# B&R Automation Studio project SiemensBRCommunication
Automation Studio 4.10.2.37; technology packages: mapp 5.12.1, mappView 5.12.1

## Configuration Config2

CPU X20CP1584, AutomationRuntime B4.91, Build 4.1.2, Safety 0.0, Vc V4.72.2

### Task classes (Cpu.sw)
```
Cyclic#4:
  Com <- Com.prg
DataObjects: comDAVCfg <- comDAVCfg.dob, comDAVMap <- comDAVMap.dob
Binaries: FWRules, udbdef, TCData, mvLoader, arconfig, User, Role, iomap, asfw, ashwac, ashwd, sysconf, vcgclass, arsvcreg
Libraries: AsTCP, sys_lib, dvframe, asstring, runtime, standard, AsMem, AsIecCon, astime, DAVNoDave, arssl, fileio, dataobj, vcresman, aruser
```

### Hardware
```
X20CP1584 : X20CP1584 v1.9.0.0
  Connector IF2:
    ActivateDevice = 1
    Mode = Manual
    InternetAddress = 192.168.0.3
    SubnetMask = 255.255.255.0
  Connector IF3:
    Operation = EthOnly
    EthernetMode = Manual
    InternetAddress = 10.42.10.220
    SubnetMask = 255.255.255.0
  ConfigurationID = komunikaceSIMATIC_Config2
  UserPartitionSize = 100
  AutomaticTransferOfUserfiles = on
  FileDevice1
  FileDeviceName1 = Flashcard
  FileDevicePath1 = C:\
  FtpUser1
  FtpUsername1 = admin
  FtpUserPassword1 = b1OGEwZ56wPH8RQzCv5cMjA1xEZ3AQeIlDvIGC2uv18=
  FtpUserSalt1 = TsE2z1/6
  FTPAccessRight1 = 0
  FTPdevice1 = ALL
  ActivateOpcUa = 1
  OpcUaInformationModels_PV_Version = 1
```

## Logical view

Binary libraries used (declarations not repeated): AsTCP, sys_lib, dvframe, asstring, runtime, standard, AsMem, AsIecCon, astime, DataObj

### Global.typ - Global data types
```iecst
TYPE
	comunicationStatus :
		(
		Initializing,
		Connecting,
		Connected,
		Disconnecting,
		Disconected,
		InitializationError,
		ConnectionError,
		ClientError,
		DisconnectingError
	);
END_TYPE
```

### Package Logical/Libraries - Global libraries

### Library Logical/Libraries/DAVNoDave (IEC, version 1.04.0) - A library based on LibNoDave to connect to a Siemens PLC
Depends on: AsTCP, DataObj, sys_lib, dvframe, asstring

#### DAVNoDave.fun - Exported functions and function blocks
```iecst
(********************************************************************
 * COPYRIGHT -- B&R Industrial Automation
 ********************************************************************
 * Library: DAVNoDave
 * File: DAVNoDave.fun
 * Author: morrisd
 * Created: May 26, 2009
 ********************************************************************
 * Functions and function blocks of library DAVNoDave
 ********************************************************************)
(**)
(*Initialization*)

FUNCTION_BLOCK DAVinitialize (*Allocates memory for communications*)
	VAR_INPUT
		enable : BOOL; (*Enable function block*)
		reset : BOOL; (*Resets the function block in case of error or if you want to reload the dataobjects ...*)
		pDOConfig : UDINT; (*Address of the name of the data object used for configuration*)
		pDOMapping : UDINT; (*Address of the name of the data object used for variable mapping*)
		pMemIdent : UDINT; (*Pointer to memory allocated by user in InitUp*)
		numItemsConfig : UINT; (*Maximum number of items in the configuration data object*)
		numItemsMapping : UINT; (*Maximum number of items in the mapping data object*)
	END_VAR
	VAR_OUTPUT
		status : UINT; (*Function block status*)
		handle : UDINT; (*Handle (for other functions)*)
	END_VAR
	VAR
		state : USINT;
		pConfig : REFERENCE TO DAVConfig_typ;
		pConfigSwap : REFERENCE TO DAVConfig_typ;
		pMapping : REFERENCE TO DAVMapping_typ;
		pMappingSwap : REFERENCE TO DAVMapping_typ;
		pDAV : REFERENCE TO DAVHandle_typ;
		pData : REFERENCE TO ARRAY[0..499] OF USINT;
		DatObjInfo_Config : DatObjInfo;
		DatObjInfo_Map : DatObjInfo;
		DatObjRead_0 : DatObjRead;
		charIdx : UDINT;
		configIdx : UINT;
		configTemp : DAVConfig_typ;
		orderIdx : UINT;
		scanCount : UDINT;
		curDataLength : UDINT;
		status_i : UINT;
		curVarType : UDINT;
		curDimensions : UDINT;
		mappingTemp : DAVMapping_typ;
		lengthToAllocate : UDINT;
		pDOData : UDINT;
		mappingIdx : UINT;
		straSplit : ARRAY[0..9] OF STRING[100];
		posNextNull : UINT;
		tmpAdr : UDINT;
		tmpVal : DINT;
		posPlus : UINT;
		memFreeFB : {REDUND_UNREPLICABLE} ARRAY[0..1] OF AsMemPartFree;
		memAllocFB : {REDUND_UNREPLICABLE} ARRAY[0..1] OF AsMemPartAllocClear;
		memHandle : {REDUND_UNREPLICABLE} ARRAY[0..1] OF UDINT;
		i : {REDUND_UNREPLICABLE} USINT;
	END_VAR
END_FUNCTION_BLOCK
(**)
(*Connection*)

FUNCTION_BLOCK DAVconnect (*Connects to a Siemens S7 or VIPA unit via ISO/TCP*)
	VAR_INPUT
		enable : BOOL; (*Enable function block*)
		pHandle : UDINT; (*Address of handle from DAVinitialize*)
		protocol : USINT; (*Connection mode. Use DAV_PROTOCOL_xxx*)
		pMPIinterface : UDINT; (*MPI interface to use (i.e. 'IF1')*)
		pMPIconnection : UDINT; (*MPI connection parameters. Use 0 for DAV_DEFAULT_MPI*)
		MPIspeed : USINT; (*MPI speed. Use DAV_SPEED_xxx*)
		MPIlocalAdr : USINT; (*MPI local address. Usually 1*)
		MPIplcAdr : USINT; (*MPI PLCl address. Usually 2*)
		pTCPsourceIP : UDINT; (*TCP ethernet interface - use 0 for listenning in on all interfaces.*)
		pTCPtargetIP : UDINT; (*TCP IP address to connect to*)
		TCPport : UINT; (*TCP port to use - use 0 for DAV_DEFAULT_PORT*)
		TCPrack : USINT; (*TCP rack number (usually 0)*)
		TCPslot : USINT; (*TCP slot number (usually 1)*)
		timeout : UINT; (*Timout time*)
	END_VAR
	VAR_OUTPUT
		status : UINT; (*Function block status*)
		pduLength : UINT; (*Length of PDU (from PLC)*)
		portOpened : UINT; (*Port number used for connection*)
		TCPident : UDINT;
	END_VAR
	VAR
		pDAV : REFERENCE TO DAVHandle_typ;
		pBufferR : REFERENCE TO ARRAY[0..99] OF USINT;
		state : USINT;
		frmConfig : XOPENCONFIG;
		FRM_xopen_0 : FRM_xopen;
		TcpOpen_0 : TcpOpen;
		TcpClient_0 : TcpClient;
		DAVexchange_0 : DAVexchange;
		TON_10ms_ClientTimeout : TON_10ms;
	END_VAR
END_FUNCTION_BLOCK

FUNCTION_BLOCK DAVdisconnect (*Disconnects current connection*)
	VAR_INPUT
		enable : BOOL; (*Enable function block*)
		pHandle : UDINT; (*Address of handle from DAVinitialize*)
		timeout : UINT;
	END_VAR
	VAR_OUTPUT
		status : UINT; (*Function block status*)
	END_VAR
	VAR
		pDAV : REFERENCE TO DAVHandle_typ;
		TcpClose_0 : TcpClose;
		FRM_close_0 : FRM_close;
		DAVexchange_0 : DAVexchange;
		state : USINT;
	END_VAR
END_FUNCTION_BLOCK
(**)
(*Servicing*)

FUNCTION_BLOCK DAVclient (*Services communcations between a B&R and Siemens PLC*)
	VAR_INPUT
		enable : BOOL; (*Enable function block*)
		pHandle : UDINT; (*Address of handle from DAVinitialize*)
		pause : BOOL; (*Pause the data transfer*)
		timeout : UINT; (*Timeout when reading*)
	END_VAR
	VAR_OUTPUT
		status : UINT; (*Function block status*)
		paused : BOOL; (*Whether the communications have been paused*)
		errorPackets : UINT; (*Number of misconfigured packets*)
		safeToDisconnect : BOOL; (*TRUE when the user can disconnect*)
	END_VAR
	VAR
		state : USINT;
		pDAV : REFERENCE TO DAVHandle_typ;
		pConfig : REFERENCE TO DAVConfig_typ;
		pMapping : REFERENCE TO DAVMapping_typ;
		ppBuffer : REFERENCE TO ARRAY[0..499] OF USINT;
		DAVexchange_0 : DAVexchange;
		currentMode : USINT;
		currentPriority : USINT;
		addIdx : UINT;
		findIdx : USINT;
		itemIdx : UINT;
		mapIdx : UINT;
		readIdx : UINT;
		numItems : USINT;
		varList : ARRAY[0..19] OF UINT;
		curValue : UDINT;
		dataLength : UINT;
		bufferFull : BOOL;
		moreLinesToScan : BOOL;
		writeValues : ARRAY[0..19] OF UDINT;
		responseSize : UINT;
		numItemsCfg : USINT;
		numItemsMap : USINT;
		maxSendSize : UINT;
		useVariable : BOOL;
		pEnable : REFERENCE TO BOOL;
	END_VAR
END_FUNCTION_BLOCK
(**)
(*Internal - Data exchange*)

FUNCTION_BLOCK DAVexchange (*Exchanges data between PLC's*)
	VAR_INPUT
		enable : BOOL; (*Enable function block*)
		pHandle : UDINT; (*Address of handle from DAVinitialize*)
		sendLength : UINT; (*Length of data to send*)
		timeout : UINT; (*Timeout when reading*)
		mpiFullExchange : BOOL; (*Full exchange of data, including Acknowledges. MPI protocol only*)
	END_VAR
	VAR_OUTPUT
		status : UINT; (*Function block status*)
		recvLength : UINT; (*Received number of bytes (not including header)*)
		recvParamLength : UINT; (*Length of parameter area*)
		recvDataLength : UINT; (*Length of data area*)
		recvStartOfDataIdx : UINT; (*Number of bytes (index 0) before data starts*)
	END_VAR
	VAR
		state : USINT;
		pDAV : REFERENCE TO DAVHandle_typ;
		ppBuffer : REFERENCE TO ARRAY[0..19] OF USINT;
		TcpSend_0 : TcpSend;
		TcpRecv_0 : TcpRecv;
		TON_10ms_Timeout : TON_10ms;
		DAVmpiSend_0 : DAVmpiSend;
		DAVmpiRead_0 : DAVmpiRead;
		bufferRead : ARRAY[0..19] OF USINT;
		bufferSend : ARRAY[0..19] OF USINT;
		sendAckNumber : USINT;
		lastState : USINT;
	END_VAR
END_FUNCTION_BLOCK

FUNCTION_BLOCK DAVmpiSend (*Sends data via serial (DVFrame library)*)
	VAR_INPUT
		enable : BOOL; (*Enable function block*)
		ident : UDINT; (*Ident from FRM_Xopen*)
		sendLength : UINT; (*Length to send*)
		pBufferW : UDINT; (*Pointer to data to send*)
	END_VAR
	VAR_OUTPUT
		status : UINT; (*Function block status*)
	END_VAR
	VAR
		FRM_gbuf_0 : FRM_gbuf;
		FRM_write_0 : FRM_write;
		FRM_robuf_0 : FRM_robuf;
	END_VAR
END_FUNCTION_BLOCK

FUNCTION_BLOCK DAVmpiRead (*Reads data via serial (DVFrame library)*)
	VAR_INPUT
		enable : BOOL; (*Enable function block*)
		ident : UDINT; (*Ident from FRM_Xopen*)
		pBufferR : UDINT; (*Maximum length to read*)
		readLength : UINT; (*Pointer to storage to read data into*)
	END_VAR
	VAR_OUTPUT
		status : UINT; (*Function block status*)
		recvBufferLength : UINT;
	END_VAR
	VAR
		FRM_read_0 : FRM_read;
		FRM_rbuf_0 : FRM_rbuf;
	END_VAR
END_FUNCTION_BLOCK
(**)
(*Internal - Packets*)

FUNCTION DAVpacketHeader : UINT (*Initializes a packet with the required protocol and TPDU. Returns the index to the start of the TPDU*)
	VAR_INPUT
		pDAV : REFERENCE TO DAVHandle_typ; (*Pointer to DAVHandle_typ*)
		pBuffer : REFERENCE TO ARRAY[0..19] OF USINT; (*Pointer to buffer to build the message*)
	END_VAR
END_FUNCTION

FUNCTION DAVpacketReadInit : UINT (*Initializes a packet for writing variables. Returns number of bytes in the buffer*)
	VAR_INPUT
		pDAV : REFERENCE TO DAVHandle_typ; (*Pointer to DAVHandle_typ*)
		pBuffer : REFERENCE TO ARRAY[0..19] OF USINT; (*Pointer to buffer to build the message*)
	END_VAR
END_FUNCTION

FUNCTION DAVpacketReadAddVar : UINT (*Adds a variable to a read packet. Returns number of bytes in the buffer*)
	VAR_INPUT
		pDAV : REFERENCE TO DAVHandle_typ; (*Pointer to DAVHandle_typ*)
		pBuffer : REFERENCE TO ARRAY[0..19] OF USINT; (*Pointer to buffer to build the message*)
		pVar : REFERENCE TO DAVSendVar_typ; (*Pointer to variable configuration to use*)
	END_VAR
	VAR
		ppBuffer : REFERENCE TO ARRAY[0..12] OF USINT;
		packetLength : UINT;
		paramLength : UINT;
	END_VAR
END_FUNCTION

FUNCTION DAVpacketWriteInit : UINT (*Initialiizes a packet for writing variables. Returns number of bytes in the buffer*)
	VAR_INPUT
		pDAV : REFERENCE TO DAVHandle_typ; (*Pointer to DAVHandle_typ*)
		pBuffer : REFERENCE TO ARRAY[0..19] OF USINT; (*Pointer to buffer to build the message*)
	END_VAR
END_FUNCTION

FUNCTION DAVpacketWriteAddVar : UINT (*Adds a variable to a write packet. Returns number of bytes in the buffer*)
	VAR_INPUT
		pDAV : REFERENCE TO DAVHandle_typ; (*Pointer to DAVHandle_typ*)
		pBuffer : REFERENCE TO ARRAY[0..19] OF USINT; (*Pointer to buffer to build the message*)
		pWriteBuffer : REFERENCE TO ARRAY[0..3] OF USINT; (*Pointer to write data*)
		pVar : REFERENCE TO DAVSendVar_typ; (*Pointer to variable configuration to use*)
	END_VAR
	VAR
		ppBuffer : REFERENCE TO ARRAY[0..12] OF USINT;
		packetLength : UINT;
		paramLength : UINT;
		dataLength : UINT;
		pBufferData : UDINT;
	END_VAR
END_FUNCTION

FUNCTION DAVpacketTCPconnect : UINT (*Creates packets for establishing a connection to a PLC via ISO/TCP. Returns number of bytes in the buffer*)
	VAR_INPUT
		pDAV : REFERENCE TO DAVHandle_typ; (*Pointer to DAVHandle_typ*)
		pBuffer : REFERENCE TO ARRAY[0..25] OF USINT; (*Pointer to buffer to build the message*)
		num : USINT; (*Packet to create*)
	END_VAR
END_FUNCTION

FUNCTION DAVpacketMPIconnect : UINT (*Creates packets for establishing a connection to a PLC via MPI. Returns number of bytes in the buffer*)
	VAR_INPUT
		pDAV : REFERENCE TO DAVHandle_typ; (*Pointer to DAVHandle_typ*)
		pBuffer : REFERENCE TO ARRAY[0..49] OF USINT; (*Pointer to buffer to build the message*)
		num : USINT; (*Packet to create*)
	END_VAR
END_FUNCTION

FUNCTION DAVpacketMPIdisconnect : UINT (*Creates packets for disconnect from a PLC via MPI. Returns number of bytes in the buffer*)
	VAR_INPUT
		pDAV : REFERENCE TO DAVHandle_typ; (*Pointer to DAVHandle_typ*)
		pBuffer : REFERENCE TO ARRAY[0..19] OF USINT; (*Pointer to buffer to build the message*)
		num : USINT; (*Packet to create*)
	END_VAR
END_FUNCTION

FUNCTION DAVpacketMPIack : UINT (*Creates packets for sending an Acknowledge to a PLC via MPI. Returns number of bytes in the buffer*)
	VAR_INPUT
		pDAV : REFERENCE TO DAVHandle_typ; (*Pointer to DAVHandle_typ*)
		pBuffer : REFERENCE TO ARRAY[0..11] OF USINT; (*Pointer to buffer to build the message*)
		ackNum : USINT; (*Acknowledge number to use*)
	END_VAR
END_FUNCTION

FUNCTION DAVresponseMPIconnect : UINT (*Compares the response of a packet from the PLC with what is expected. Returns if the packet is okay*)
	VAR_INPUT
		pDAV : REFERENCE TO DAVHandle_typ; (*Pointer to DAVHandle_typ*)
		pBuffer : REFERENCE TO ARRAY[0..49] OF USINT; (*Pointer to buffer to compare the message*)
		num : USINT; (*Packet to compare*)
	END_VAR
END_FUNCTION
(**)
(*Internal - Swap bytes*)

FUNCTION DAVswapWORD : UINT (*Swaps bytes in a WORD*)
	VAR_INPUT
		pUINT : REFERENCE TO UINT; (*Address of UINT variable*)
	END_VAR
END_FUNCTION

FUNCTION DAVswapDWORD : UDINT (*Swaps bytes and words in a DWORD*)
	VAR_INPUT
		pUDINT : REFERENCE TO UDINT; (*Address of UDINT variable*)
	END_VAR
END_FUNCTION
(**)
(*Internal - Get bytes*)

FUNCTION DAVgetHIBYTE : USINT (*Returns the hi-byte from a WORD*)
	VAR_INPUT
		input : UINT; (*Input WORD*)
	END_VAR
END_FUNCTION

FUNCTION DAVgetLOBYTE : USINT (*Returns the lo-byte from a WORD*)
	VAR_INPUT
		input : UINT; (*Input WORD*)
	END_VAR
END_FUNCTION

FUNCTION DAVaddressBITS : USINT (*Returns a byte of the start address*)
	VAR_INPUT
		startAdr : UDINT; (*Start address of variable*)
		byteNum : USINT; (*Byte number to return*)
	END_VAR
END_FUNCTION
(**)
(*Internal - Combine bytes*)

FUNCTION DAVmakeWORD : UINT (*Returns a WORD from 2 bytes*)
	VAR_INPUT
		hiByte : USINT; (*Hi-byte input*)
		loByte : USINT; (*Lo-byte input*)
	END_VAR
END_FUNCTION

FUNCTION DAVupdateVAR : USINT (*Updates the selected variable*)
	VAR_INPUT
		pMapping : REFERENCE TO DAVMapping_typ; (*Pointer to a DAVMapping_typ*)
		pBuffer : UDINT; (*Address of buffer to read the value*)
		transportBOOL : BOOL; (*Transport mechanism for BOOLEAN data*)
	END_VAR
	VAR
		pDynBool : REFERENCE TO BOOL;
		pDynByte : REFERENCE TO USINT;
		pDynWord : REFERENCE TO UINT;
		pDynDWord : REFERENCE TO UDINT;
		tempVar : UDINT;
	END_VAR
END_FUNCTION

FUNCTION DAVcalcVARadr : USINT
	VAR_INPUT
		pVar : REFERENCE TO DAVSendVar_typ; (*Pointer to DAVSendVar_typ*)
	END_VAR
	VAR
		pUserDB : REFERENCE TO UINT;
		pUserStartAdr : REFERENCE TO UINT;
		pUserStartAdrB : REFERENCE TO USINT;
	END_VAR
END_FUNCTION
(**)
(*Internal - Misc*)

FUNCTION DAVsplit : UINT
	VAR_INPUT
		pData : UDINT; (*Address of data to read*)
		pSplitData : REFERENCE TO ARRAY[0..9] OF STRING[100]; (*Pointer to array of strings*)
	END_VAR
	VAR
		ppData : REFERENCE TO ARRAY[0..499] OF USINT;
		ppSplitData : REFERENCE TO ARRAY[0..99] OF USINT;
		splitIdx : USINT;
		charIdx : UINT;
		copyIdx : UINT;
	END_VAR
END_FUNCTION

FUNCTION DAVisnumeric : BOOL
	VAR_INPUT
		pString : UDINT; (*Pointer to string to compare*)
	END_VAR
	VAR
		pData : REFERENCE TO ARRAY[0..99] OF USINT;
		charIdx : USINT;
	END_VAR
END_FUNCTION

FUNCTION DAVmpiCalcCS : BOOL
	VAR_INPUT
		pBuffer : REFERENCE TO ARRAY[0..99] OF USINT; (*Address of buffer*)
		len : UINT; (*Length to data*)
	END_VAR
	VAR
		charIdx : UINT;
		checksum : USINT;
	END_VAR
END_FUNCTION

FUNCTION DAVmpiSuffixCRC : UINT (*Performs DLE doubling, adds DLE and ETX and BCC (checksum)*)
	VAR_INPUT
		pBuffer : REFERENCE TO ARRAY[0..499] OF USINT; (*Pointer to buffer to build the message*)
		len : UINT; (*Length of data in the buffer*)
	END_VAR
	VAR
		bufferR : ARRAY[0..499] OF USINT;
		sourceIdx : UINT;
		destIdx : UINT;
		bcc : USINT;
	END_VAR
END_FUNCTION

FUNCTION DAVdecodeMPI : UINT (*Removes DLE doubling from a received message*)
	VAR_INPUT
		pBuffer : REFERENCE TO ARRAY[0..499] OF USINT; (*Pointer to buffer which contains the message*)
		bufferSize : UINT; (*Total size of the buffer*)
		dataLength : UINT; (*Length of data currently in the buffer*)
	END_VAR
	VAR
		bufferOrig : ARRAY[0..499] OF USINT;
		sourceIdx : UINT;
		destIdx : UINT;
	END_VAR
END_FUNCTION
```

#### DAVNoDave.typ - Exported data types
```iecst
(********************************************************************
 * COPYRIGHT -- B&R Industrial Automation
 ********************************************************************
 * Library: DAVNoDave
 * File: DAVNoDave.typ
 * Author: morrisd
 * Created: May 26, 2009
 ********************************************************************
 * Functions and function blocks of library DAVNoDave
 ********************************************************************)
(**)
(*DAV Handle*)

TYPE
	DAVHandle_typ : 	STRUCT  (*Main DAVNoDave structure*)
		connection : DAVHandleConnect_typ; (*Connection data*)
		ident : UDINT; (*Identity for TCP / MPI comms*)
		pConfig : UDINT; (*Address of comms configuration*)
		pMapping : UDINT; (*Address of mapping configuration*)
		pBufferR : UDINT; (*Address of read buffer*)
		pBufferW : UDINT; (*Address of write buffer*)
		internal : USINT; (*Internal*)
		maxLinesConfig : UINT; (*Maximum number of lines in configuration*)
		maxLinesMapping : UINT; (*Maximum number of lines in mapping*)
		maxPrioirty : USINT; (*Maximum prioirty level found in the configuration data object*)
	END_STRUCT;
	DAVHandleConnect_typ : 	STRUCT  (*DAVNoDave communications*)
		protocol : USINT; (*Protocol (DAV_PROTOCOL_xxx)*)
		mpiSpeed : USINT; (*MPI speed (DAV_SPEED_xxx)*)
		mpiLocalAdr : USINT; (*MPI local address (usually 1)*)
		mpiPLCAdr : USINT; (*MPI PLC address (usually 2)*)
		tcpRack : USINT; (*TCP rack*)
		tcpSlot : USINT; (*TCP slot*)
		connectNum : USINT; (*MPI connection number*)
		connectNum2 : USINT; (*MPI connection number 2*)
		msgNum : USINT; (*Packet number*)
		pduNum : UINT; (*PDU number*)
		ackNum : USINT; (*Acknowledge number*)
	END_STRUCT;
END_TYPE

(**)
(*Data Object (per line)*)

TYPE
	DAVSendVar_typ : 	STRUCT  (*Structure per variable per variable*)
		area : USINT; (*Siemens - Area (DAV_AREA_xxx)*)
		db : UINT; (*Siemens - Data block number (only if area is DAV_AREA_DB)*)
		pdb : UDINT; (*Siemens - Pointer to Data block number (only if area is DAV_AREA_DB)*)
		actAdr : UINT; (*Siemens - Actual variable address (in BYTE's)*)
		bitAdr : UDINT; (*Siemens - Start address (in BIT's)*)
		pStartAdr : UDINT; (*Siemens - Pointer to Start address (must be a UINT)*)
		bitAdrB : USINT; (*Siemens - Start address bit position*)
		pStartAdrB : UDINT; (*Siemens - Pointer to start address bit position (must be a USINT)*)
		type : USINT; (*Siemens - Variable type (DAV_VAR_xxx)*)
		length : UINT; (*Siemens - Variable length*)
	END_STRUCT;
	DAVConfig_typ : 	STRUCT  (*Structure per line in the configuration data object*)
		var : DAVSendVar_typ; (*Variable details*)
		priority : USINT; (*Priority of variable*)
		pEnable : UDINT; (*Pointer to enable variable (must be a BOOL)*)
		brVarAdr : UDINT; (*B&R - Start address of variable(s)*)
		internal : USINT; (*Internal variable*)
	END_STRUCT;
	DAVMapping_typ : 	STRUCT  (*Structure per line in the mapping data object*)
		var : DAVSendVar_typ; (*Variable details*)
		priority : USINT; (*Priority of variable*)
		pEnable : UDINT; (*Pointer to enable variable (must be a BOOL)*)
		access : USINT; (*Access (0 = read, 1= write, 2 = both)*)
		brVarAdr : UDINT; (*B&R - Address of variable to store the value*)
		brVarLength : USINT; (*B&R - Length of variable*)
		brVarType : USINT; (*B&R - Variable type*)
		brPrevValue : UDINT; (*B&R - Previous value*)
		internal : USINT; (*Internal variable*)
		cfgIndex : UINT; (*Internal configuration index*)
	END_STRUCT;
END_TYPE
```

#### DAVNoDave.var - Exported constants
```iecst
(********************************************************************
 * COPYRIGHT -- B&R Industrial Automation
 ********************************************************************
 * Library: DAVNoDave
 * File: DAVNoDave.var
 * Author: morrisd
 * Created: May 26, 2009
 ********************************************************************
 * Constants of library DAVNoDave
 ********************************************************************)
(**)
(*Internal*)
VAR CONSTANT
	DAV_DEFAULT_BUFFER_R : UINT := 500; (*Default read buffer size, should be more than PDU size*)
	DAV_DEFAULT_BUFFER_W : UINT := 500; (*Default write buffer size, should be more than PDU size*)
END_VAR
(**)
(*Default values*)
VAR CONSTANT
	DAV_DEFAULT_SOURCE_PORT : UINT := 60000; (*Default source port (should be >=49152)*)
	DAV_DEFAULT_PORT : UINT := 102; (*Default connection port*)
	DAV_DEFAULT_MPI : STRING[40] := '/PHY=RS232 /BD=38400 /PA=O /DB=8 /SB=1'; (*Default connection for MPI*)
	DAV_DEFAULT_TIMEOUT : UINT := 0; (*Default timeout (1500ms for ISO/TCP, 5000ms for MPI)*)
END_VAR
(**)
(*Configuration*)
VAR CONSTANT
	DAV_CONFIG_MAX_LINES : UINT := 500; (*Maximum number of lines in the configuration file*)
	DAV_CONFIG_PRIOIRTY_MAX : USINT := 5; (*Prioirty level (maximum)*)
	DAV_CONFIG_RW_B : USINT := 2; (*Access level (read / write)*)
	DAV_CONFIG_RW_R : USINT := 1; (*Access level (read only)*)
	DAV_CONFIG_RW_W : USINT := 3; (*Access level (write only)*)
END_VAR
(**)
(*Protocol*)
VAR CONSTANT
	DAV_PROTOCOL_TCP : USINT := 100; (*Connection type - ISOTCP*)
	DAV_PROTOCOL_MPI : USINT := 200; (*Connection type - MPI*)
END_VAR
(**)
(*Protocol - Speed*)
VAR CONSTANT
	DAV_SPEED_9K : USINT := 0; (*MPI Adapter speed - 9k baud*)
	DAV_SPEED_19K : USINT := 1; (*MPI Adapter speed - 19k baud*)
	DAV_SPEED_187K : USINT := 2; (*MPI Adapter speed - 187k baud*)
	DAV_SPEED_500K : USINT := 3; (*MPI Adapter speed - 500k baud*)
	DAV_SPEED_1500K : USINT := 4; (*MPI Adapter speed - 1500k baud*)
	DAV_SPEED_45K : USINT := 5; (*MPI Adapter speed - 45k baud*)
	DAV_SPEED_93K : USINT := 6; (*MPI Adapter speed - 93k baud*)
END_VAR
(**)
(*PDU Constants*)
VAR CONSTANT
	DAV_PDU_SIZE : UINT := 240; (*PDU size*)
END_VAR
(**)
(*Variables*)
VAR CONSTANT
	DAV_VAR_BIT : USINT := 1; (*Read a single bit*)
	DAV_VAR_BYTE : USINT := 2; (*Read a byte*)
	DAV_VAR_WORD : USINT := 4; (*NOT IMPLEMENTED Read a word*)
END_VAR
(**)
(*DataBlock's and Area*)
VAR CONSTANT
	DAV_AREA_COUNTER : USINT := 28; (*NOT IMPLEMENTED Area type, S7 Counters*)
	DAV_AREA_DB : USINT := 132; (*Area type, DataBlocks*)
	DAV_AREA_DI : USINT := 133; (*NOT IMPLEMENTED Area type, DataBlock Instance*)
	DAV_AREA_FLAG : USINT := 131; (*Area type, Flags*)
	DAV_AREA_INPUT : USINT := 129; (*Area type, Inputs*)
	DAV_AREA_LOCAL : USINT := 134; (*NOT IMPLEMENTED Area type, Local (not tested)*)
	DAV_AREA_OUTPUT : USINT := 130; (*Area type, Outputs*)
	DAV_AREA_PERIPHERAL : USINT := 128; (*NOT IMPLEMENTED Area type, Peripherals*)
	DAV_AREA_TIMER : USINT := 29; (*NOT IMPLEMENTED Area type, S7 Timers*)
END_VAR
(**)
(*Error codes*)
VAR CONSTANT
	DAV_ERR_INITIALIZATION : UINT := 51000; (*Initialization error*)
	DAV_ERR_HANDLE : UINT := 51001; (*Invalid handle specified*)
	DAV_ERR_BUFFER : UINT := 51002; (*Invalid buffer specified*)
	DAV_ERR_BUFFER_SIZE : UINT := 51003; (*Invalid buffer size specified*)
	DAV_ERR_CONNECT_OPEN : UINT := 51004; (*Connection already open*)
	DAV_ERR_CONNECT_CLOSED : UINT := 51005; (*Connection already closed*)
	DAV_ERR_CONNECT_PROTOCOL : UINT := 51006; (*Invalid connection mode specidied*)
	DAV_ERR_CONNECT_TARGETIP : UINT := 51007; (*Invalid target IP specified*)
	DAV_ERR_CONNECT_INTERFACE : UINT := 51008; (*Invalid interface specified*)
	DAV_ERR_CONNECT_TCP : UINT := 51009; (*Can not connect to specified TCP/IP address*)
	DAV_ERR_SEND_MISSINGDATA : UINT := 51010; (*Not all the data was sent*)
	DAV_ERR_SEND_NODATA : UINT := 51011; (*Invalid send length*)
	DAV_ERR_SEND_BUFFERSIZE : UINT := 51012; (*Buffer size too small*)
	DAV_ERR_RECV_NODATA : UINT := 51020; (*No data received - client disconnect?*)
	DAV_ERR_RECV_MISSINGDATA : UINT := 51021; (*Not all the data was received*)
	DAV_ERR_RECV_WRONGPACKET : UINT := 51022; (*Wrong packet received*)
	DAV_ERR_RECV_BUFFERSIZE : UINT := 51023; (*Buffer size too small*)
	DAV_ERR_RECV_PROTOCOL : UINT := 51024; (*MPI protocol error*)
	DAV_ERR_RECV_RESPONSE : UINT := 51025; (*MPI response*)
	DAV_ERR_FAILED_READ : UINT := 51027; (*Failed to read data*)
	DAV_ERR_FAILED_WRITE : UINT := 51028; (*Failed to write data*)
	DAV_ERR_TIMEOUT : UINT := 51029; (*Timeout occured*)
	DAV_ERR_CFG_DONAME : UINT := 51030; (*Invalid configuration specified*)
	DAV_ERR_CFG_DONODATA : UINT := 51031; (*Invalid configuration data (none available)*)
	DAV_ERR_CFG_INVALID : UINT := 51032; (*Invalid configuration data*)
	DAV_ERR_CFG_MAXLINES : UINT := 51033; (*Invalid number of lines specified*)
	DAV_ERR_CFG_TIMEOUT : UINT := 51034; (*Execution too long*)
	DAV_ERR_MPI_ADAPTER : UINT := 51040; (*Unsupported MPI adapter*)
	DAV_ERR_ACKNOWLEDGE : UINT := 51041;
END_VAR
```

#### DAVinitialize.st - Initializes data object(s) for servicing communications
```iecst
(********************************************************************************************************************************)
(* COPYRIGHT -- B&R Industrial Automation																																												*)
(********************************************************************************************************************************)
(* Library:				DAVNoDave																																																			*)
(* File: 					DAVinitialize.st																																															*)
(* Author: 				morrisd																																																				*)
(* Created: 			May 26, 2009																																																	*)
(********************************************************************************************************************************)

(********************************************************************************************************************************)
(* DAVinitialize																																																								*)
(*==============================================================================================================================*)
(* Initializes the configuration object to communicate between the PLC and the Siemen's PLC																			*)
(* Note:																																																												*)
(*			1) This function needs to be called in the INIT program. 																																*)
(*			2) It should be called once and not continously in a loop (as we call it in a loop).																		*)
(* Returns a status																																																							*)
(********************************************************************************************************************************)
FUNCTION_BLOCK DAVinitialize

	(* Function not enabled *)
	IF(enable = FALSE)THEN
		status := 65534;

	(* Invalid data object *)
	ELSIF((pDOConfig = 0) AND (numItemsConfig > 0))THEN
 		status:= DAV_ERR_CFG_DONAME;

	(* Invalid data object *)
	ELSIF(pDOMapping = 0)THEN
 		status:= DAV_ERR_CFG_DONAME;

 	(* Invalid number of items *)
	ELSIF((numItemsConfig > DAV_CONFIG_MAX_LINES) OR (numItemsMapping > DAV_CONFIG_MAX_LINES))THEN
 		status:= DAV_ERR_CFG_MAXLINES;

	(* Run the function *)
	ELSE
			(* Error occured *)
			IF status <> 65535 AND status <> ERR_OK AND state < 255 THEN
				state := 255;
			END_IF

			(**************************************************************************************************************************)
			(* Function Operation                                                                   																	*)
			(**************************************************************************************************************************)
			CASE state OF

				(************************************************************************************************************************)
				(* InitStuff		               																															*)
				(************************************************************************************************************************)
				0:
					(* Reset handle *)
					handle:= 0;
					(* Reset our internal counter *)
					scanCount:= 0;
					(* Make status busy *)
					status:= 65535;
					state:= 1;

				(************************************************************************************************************************)
				(* Get DataObject Information - pDOConfig		               																															*)
				(************************************************************************************************************************)
				1:

					(* Config Data Object Enabled *)
					IF(numItemsConfig > 0)THEN

						(* Get information *)
						DatObjInfo_Config.enable:=		TRUE;										(* Enable function block *)
						DatObjInfo_Config.pName:=			pDOConfig;							(* Pointer to Data Object name *)
						DatObjInfo_Config();																(* Service the function block *)
						scanCount:= scanCount + 1;
						IF ((DatObjInfo_Config.status <> 65535) OR (scanCount > 10000)) THEN

							(* Complete *)
							IF((DatObjInfo_Config.status = 0) AND (DatObjInfo_Config.len > 0))THEN
								scanCount := 0;
								state:= 2;

							(* Invalid length *)
							ELSIF(DatObjInfo_Config.status = 0)THEN
								status:= DAV_ERR_CFG_DONODATA;

							(* Timeout *)
							ELSIF(DatObjInfo_Config.status = 65535)THEN
								status:= DAV_ERR_CFG_TIMEOUT;

							(* Error *)
							ELSE
								status:= DatObjInfo_Config.status;
							END_IF

						END_IF

					(* Config Data Object Disabled *)
					ELSE
						state:= 2;
					END_IF
				(************************************************************************************************************************)

				(************************************************************************************************************************)
				(* Get DataObject Information - pDOMapping                 																															*)
				(************************************************************************************************************************)
				2:
					(* Get information *)
					DatObjInfo_Map.enable:=				TRUE;										(* Enable function block *)
					DatObjInfo_Map.pName:=				pDOMapping;							(* Pointer to Data Object name *)
					DatObjInfo_Map();																		(* Service the function block *)
					scanCount:= scanCount + 1;
					IF ((DatObjInfo_Map.status <> 65535) OR (scanCount > 100000)) THEN

						(* Complete *)
						IF((DatObjInfo_Map.status = 0) AND (DatObjInfo_Map.len > 0))THEN
							scanCount := 0;
							state:= 5;

						(* Invalid length *)
						ELSIF(DatObjInfo_Map.status = 0)THEN
							status:= DAV_ERR_CFG_DONODATA;

						(* Timeout *)
						ELSIF(DatObjInfo_Map.status = 65535)THEN
							status:= DAV_ERR_CFG_TIMEOUT;

						(* Error *)
						ELSE
							status:= DatObjInfo_Map.status;
						END_IF

					END_IF
				(************************************************************************************************************************)

				(************************************************************************************************************************)
				(* Free all previous memory                 																															*)
				(************************************************************************************************************************)
				5: // If no MemHandle passed -> not using live allocation
					IF pMemIdent <> 0 THEN
						state := 10;
						FOR i := 0 TO SIZEOF(memHandle)/SIZEOF(memHandle[0]) - 1 DO
							(* Memory was allocated earlier *)
							IF memHandle[i] <> 0 THEN
								memFreeFB[i](enable := TRUE, ident:=pMemIdent, mem:=memHandle[i]);
								status_i := memFreeFB[i].status;
							END_IF
							IF status_i <> 0 THEN
								state := 255;
								status := memFreeFB[i].status;
								EXIT;
							END_IF
						END_FOR
						state := 10;
					ELSE
						state := 10;
					END_IF

				(************************************************************************************************************************)
				(* Allocate memory for DAVNoDave library				                   																											*)
				(************************************************************************************************************************)
				10:
					(* Determine length and allocate *)
					lengthToAllocate:=							SIZEOF(pDAV) + 														(* DAV strucutre.. *)
		 																			(numItemsConfig * SIZEOF(pConfig)) +			(* Commms configuration.. *)
										 											(numItemsMapping * SIZEOF(pMapping)) +		(* Mapping configuration.. *)
																					DAV_DEFAULT_BUFFER_R +										(* Read buffer.. *)
																					DAV_DEFAULT_BUFFER_W; 										(* Write buffer *)

					IF pMemIdent = 0 THEN (* old style *)
						status_i:= TMP_alloc(lengthToAllocate, ADR(handle));

					ELSE (* new flexible style *)
						memAllocFB[0](enable:=TRUE,	ident:=pMemIdent, len:=lengthToAllocate);
						status_i:=memAllocFB[0].status;
						IF status_i = 0 THEN
							memHandle[0] := memAllocFB[0].mem;
							handle := memAllocFB[0].mem;
						END_IF
					END_IF
					//memAllocFB[0](enable:=FALSE);

					(* Complete *)
					IF(status_i = 0)THEN

						(* Clear data, if old style is used *)
						IF pMemIdent = 0 THEN
							memset(handle, 0, lengthToAllocate);
						END_IF

						(* Access pDAV and store the addresses *)
						pDAV ACCESS handle;
						pDAV.pConfig:= handle + SIZEOF(pDAV);
						pDAV.pMapping:= pDAV.pConfig + (numItemsConfig * SIZEOF(pConfig));
						pDAV.pBufferR:= pDAV.pMapping + (numItemsMapping * SIZEOF(pMapping));
						pDAV.pBufferW:= pDAV.pBufferR + DAV_DEFAULT_BUFFER_R;
						pDAV.maxLinesConfig:= 0;
						pDAV.maxLinesMapping:= 0;
						pDAV.ident:= 0;
						pDAV.internal:= 0;
						memset(ADR(pDAV.connection), 0, SIZEOF(pDAV.connection)); (* ? *)

						(* Access pConfig and pMapping *)
						pConfig ACCESS pDAV.pConfig;
						pMapping ACCESS pDAV.pMapping;

						state:= 11;

					(* Error *)
					ELSE
						status:= status_i;
					END_IF
				(************************************************************************************************************************)

				(************************************************************************************************************************)
				(* Allocate memory for reading the Data Objects            																															*)
				(************************************************************************************************************************)
				11:
					(* Determine length and allocate *)
					lengthToAllocate:=	MAX(DatObjInfo_Config.len, DatObjInfo_Map.len);		(* Length to create *)

					IF pMemIdent = 0 THEN (* old style *)
						status_i:= TMP_alloc(lengthToAllocate, ADR(pDOData));
					ELSE (* new flexible style *)
						memAllocFB[1](enable:=TRUE,	ident:=pMemIdent, len:=lengthToAllocate);
						status_i:=memAllocFB[1].status;
						IF status_i = 0 THEN
							memHandle[1] := memAllocFB[1].mem;
							pDOData := memAllocFB[1].mem;
						END_IF
					END_IF
					//memAllocFB[1](enable:=FALSE);

					(* Complete *)
					IF(status_i = 0)THEN
						(* Clear data *)
						memset(pDOData, 0, lengthToAllocate);
						IF(numItemsConfig > 0)THEN
							state:= 20;								(* Read configuration *)
						ELSE
							state:= 30;								(* Read mapping *)
						END_IF

					(* Error *)
					ELSE
						status:= status_i;
					END_IF
				(************************************************************************************************************************)

				(************************************************************************************************************************)
				(* Read configuration from the specified DataObject        																															*)
				(************************************************************************************************************************)
				20:
					(* Read user's configuration *)
					DatObjRead_0.enable:= TRUE;										(* Enable the function block *)
					DatObjRead_0.ident:= DatObjInfo_Config.ident;					(* Use the DataObj's identity *)
					DatObjRead_0.Offset:= 0;										(* Start from the beginning *)
					DatObjRead_0.pDestination:= pDOData;							(* Read data into DRAM *)
					DatObjRead_0.len:= DatObjInfo_Config.len;						(* Read the entire size of the DO *)
					DatObjRead_0();
					scanCount:= scanCount + 1;
					IF (DatObjRead_0.status <> 65535) OR (scanCount > 100000) THEN
						(* Complete *)
						IF(DatObjRead_0.status = 0)THEN
							scanCount := 0;
							(* Reset offsets *)
							charIdx:= 0;
							configIdx:= 0;
							state:= 21;

						(* Timeout *)
						ELSIF(DatObjRead_0.status = 65535)THEN
							status:= DAV_ERR_CFG_TIMEOUT;

						(* Error *)
						ELSE
							status:= DatObjRead_0.status;
						END_IF
					END_IF
				(************************************************************************************************************************)

				(************************************************************************************************************************)
				(* Create our configuration								                 																															*)
				(************************************************************************************************************************)
				21:

					(* Access next 500 characters *)
					pData ACCESS (pDOData + charIdx);

					(* Access configuration *)
					pConfig ACCESS pDAV.pConfig + (configIdx * SIZEOF(pConfig));

					(* Internal *)
					pConfig.brVarAdr:= 0;
					pConfig.internal:= 0;
					pConfig.pEnable:= 0;
					pConfig.var.pdb:= 0;
					pConfig.var.pStartAdr:= 0;
					pConfig.var.pStartAdrB:= 0;
					pConfig.var.bitAdrB:= 0;

					(* Split data *)
					(* Note: the data should be in the following format *)
					(*	[0]		-		Priority (1-5)														*)
					(*	[1]		-		Enable flag (0 for always enabled)				*)
					(*	[2]		-		Area (M, D, I, O)													*)
					(*	[3]		-		DataBlock Number (0-65535)								*)
					(*	[4]		-		Start Address (numeric)										*)
					(*	[5]		-		Length 																		*)
					(*	[6]		-		NULL																			*)
					posNextNull:= DAVsplit(ADR(pData), ADR(straSplit));

					(* Ensure we have a valid NULL *)
					IF((posNextNull > 0) AND
						(strlen(ADR(straSplit[0])) > 0) AND
						(strlen(ADR(straSplit[1])) > 0) AND
						(strlen(ADR(straSplit[2])) > 0) AND
						(strlen(ADR(straSplit[3])) > 0) AND
						(strlen(ADR(straSplit[4])) > 0) AND
						(strlen(ADR(straSplit[5])) > 0))THEN

						(* Priority *)
						tmpVal:= atoi(ADR(straSplit[0]));
						IF((tmpVal >= 1) AND (tmpVal <= USINT_TO_DINT(DAV_CONFIG_PRIOIRTY_MAX)))THEN
							pConfig.priority:= DINT_TO_USINT(tmpVal);
							pDAV.maxPrioirty:= MAX(pDAV.maxPrioirty, pConfig.priority);
						ELSE
							status:= 101;
						END_IF

						(* Enable flag (either 0 or variable) *)
						IF(strcmp(ADR(straSplit[1]), ADR('0')) <> 0)THEN
							tmpAdr:= 0;
							curDataLength:= 0;
							status_i:= PV_xgetadr(ADR(straSplit[1]), ADR(tmpAdr), ADR(curDataLength));
							IF((status_i = 0) AND (tmpAdr <> 0) AND (curDataLength = 1))THEN
								pConfig.pEnable:= tmpAdr;
							ELSE
								status:= 102;
							END_IF
						END_IF

						(* Area *)
						IF(strcmp(ADR(straSplit[2]), ADR('D')) = 0)THEN
							pConfig.var.area:= DAV_AREA_DB;
						ELSIF(strcmp(ADR(straSplit[2]), ADR('M')) = 0)THEN
							pConfig.var.area:= DAV_AREA_FLAG;
						ELSIF(strcmp(ADR(straSplit[2]), ADR('I')) = 0)THEN
							pConfig.var.area:= DAV_AREA_INPUT;
						ELSIF(strcmp(ADR(straSplit[2]), ADR('O')) = 0)THEN
							pConfig.var.area:= DAV_AREA_OUTPUT;
						ELSE
							status:= 103;
						END_IF

						(* DataBlock number *)
						IF(pConfig.var.area <> DAV_AREA_DB)THEN
							pConfig.var.db:= 0;
						ELSE
							IF(DAVisnumeric(ADR(straSplit[3])) = TRUE)THEN
								tmpVal:= atoi(ADR(straSplit[3]));

								IF((tmpVal >= 0) AND (tmpVal <= 65535))THEN
									pConfig.var.db:= DINT_TO_UINT(tmpVal);
								ELSE
									status:= 104;
								END_IF
							ELSE
								tmpAdr:= 0;
								curDataLength:= 0;
								status_i:= PV_xgetadr(ADR(straSplit[3]), ADR(tmpAdr), ADR(curDataLength));
								IF((status_i = 0) AND (tmpAdr <> 0) AND (curDataLength = 2))THEN
									pConfig.var.pdb:= tmpAdr;
								ELSE
									status:= 105;
								END_IF
							END_IF
						END_IF

						(* Start address (either value or variable) *)
						IF(DAVisnumeric(ADR(straSplit[4])) = TRUE)THEN
			 				pConfig.var.actAdr:= DINT_TO_UINT(atoi(ADR(straSplit[4])));
						ELSE
							pConfig.var.actAdr:= 0;
							tmpAdr:= 0;
							curDataLength:= 0;
							status_i:= PV_xgetadr(ADR(straSplit[4]), ADR(tmpAdr), ADR(curDataLength));
							IF((status_i = 0) AND (tmpAdr <> 0) AND (curDataLength = 2))THEN
								pConfig.var.pStartAdr:= tmpAdr;
							ELSE
								status:= 106;
							END_IF
						END_IF

						(* Determine address in bits *)
						(* Note: if (pStartAdrXX > 0) then we need to keep recalculating this *)
						DAVcalcVARadr(ADR(pConfig.var));

						(* Length *)
						tmpVal:= atoi(ADR(straSplit[5]));
						IF((tmpVal > 0) AND (tmpVal < 240))THEN
			 				pConfig.var.length:= DINT_TO_USINT(tmpVal);
						ELSE
							status:= 107;
						END_IF

						pConfig.var.type:= DAV_VAR_BYTE;													(* Variable type *)
						configIdx:= configIdx + 1;															(* Use next configuration *)
						charIdx:= charIdx + posNextNull + 1;												(* Point to next line (nullIdx + 1) *)

						(* Reached number of configurations, or length of DataObject *)
						(* Note: Data Object aligns to 4 bytes *)
						IF((configIdx >= numItemsConfig) OR (charIdx >= DatObjInfo_Config.len - 4))THEN
							pDAV.maxLinesConfig:= configIdx;
							(* Clear memory *)
							memset(pDOData, 0, lengthToAllocate);									(* Number of lines used *)
							scanCount := 0;
							state:= 30;
						END_IF
					ELSE
						status:= 108;
					END_IF

					(* Error occured *)
					IF(status <> 65535)THEN
						state:= 255;
					END_IF
				(************************************************************************************************************************

				(************************************************************************************************************************)
				(* Read mapping from the specified DataObject        																																		*)
				(************************************************************************************************************************)
				30:
					(* Read user's configuration *)
					DatObjRead_0.enable:= TRUE;					(* Enable the function block *)
					DatObjRead_0.ident:= DatObjInfo_Map.ident;	(* Use the DataObj's identity *)
					DatObjRead_0.Offset:= 0;					(* Start from the beginning *)
					DatObjRead_0.pDestination:= pDOData;		(* Read data into DRAM *)
					DatObjRead_0.len:= DatObjInfo_Map.len;		(* Read the entire size of the DO *)
					DatObjRead_0();																								(* Service the function block *)
					scanCount:= scanCount + 1;

					IF (DatObjRead_0.status <> 65535) OR (scanCount > 100000) THEN
						(* Complete *)
						IF(DatObjRead_0.status = 0)THEN

							(* Reset offsets *)
							charIdx:= 0;
							configIdx:= 0;
							state:= 31;

						(* Timeout *)
						ELSIF(DatObjRead_0.status = 65535)THEN
							status:= DAV_ERR_CFG_TIMEOUT;

						(* Error *)
						ELSE
							status:= DatObjRead_0.status;
						END_IF
					END_IF
				(************************************************************************************************************************)

				(************************************************************************************************************************)
				(* Create our mapping											                 																															*)
				(************************************************************************************************************************)
				31:

					(* Access next 500 characters *)
					pData ACCESS (pDOData + charIdx);

					(* Access configuration *)
					pMapping ACCESS pDAV.pMapping + (configIdx * SIZEOF(pMapping));

					(* Internal *)
					pMapping.internal:= 0;
					pMapping.cfgIndex:= 65535;
					pMapping.pEnable:= 0;
					pMapping.var.pdb:= 0;
					pMapping.var.pStartAdr:= 0;
					pMapping.var.pStartAdrB:= 0;

					(* Split data *)
					(* Note: the data should be in the following format *)
					(*	[0]		-		Priority (1-5)														*)
					(*	[1]		-		Enable flag (0 for always enabled)				*)
					(*	[2]		-		R/W Access (W, R, B)											*)
					(*	[3]		-		Area (M, D, I, O)													*)
					(*	[4]		-		DataBlock Number (0-65535)								*)
					(*	[5]		-		Start Address (numeric or variable				*)
					(*	[6]		-		Start Address bit (numeric or variable)		*)
					(*	[7]		-		Length 																		*)
					(*	[8]		-		B&R variable name													*)
					(*	[9]		-		NULL																			*)
					posNextNull:= DAVsplit(ADR(pData), ADR(straSplit));

					(* Ensure we have a valid NULL *)
					IF((posNextNull > 0) AND
						(strlen(ADR(straSplit[0])) > 0) AND
						(strlen(ADR(straSplit[1])) > 0) AND
						(strlen(ADR(straSplit[2])) > 0) AND
						(strlen(ADR(straSplit[3])) > 0) AND
						(strlen(ADR(straSplit[4])) > 0) AND
						(strlen(ADR(straSplit[5])) > 0) AND
						(strlen(ADR(straSplit[6])) > 0) AND
						(strlen(ADR(straSplit[7])) > 0) AND
						(strlen(ADR(straSplit[8])) > 0))THEN

						(* Priority *)
						tmpVal:= atoi(ADR(straSplit[0]));
						IF((tmpVal >= 1) AND (tmpVal <= USINT_TO_DINT(DAV_CONFIG_PRIOIRTY_MAX)))THEN
							pMapping.priority:= DINT_TO_USINT(tmpVal);
							pDAV.maxPrioirty:= MAX(pDAV.maxPrioirty, pMapping.priority);
						ELSE
							status:= 109;
						END_IF

						(* Enable flag (either 0 or variable) *)
						pMapping.pEnable:= 0;
						IF(strcmp(ADR(straSplit[1]), ADR('0')) <> 0)THEN
							tmpAdr:= 0;
							curDataLength:= 0;
							status_i:= PV_xgetadr(ADR(straSplit[1]), ADR(tmpAdr), ADR(curDataLength));
							IF((status_i = 0) AND (tmpAdr <> 0) AND (curDataLength = 1))THEN
								pMapping.pEnable:= tmpAdr;
							ELSE
								status:= 110;
							END_IF
						END_IF

						(* R/W Access *)
						IF(strcmp(ADR(straSplit[2]), ADR('W')) = 0)THEN
							pMapping.access:= DAV_CONFIG_RW_W;
						ELSIF(strcmp(ADR(straSplit[2]), ADR('B')) = 0)THEN
							pMapping.access:= DAV_CONFIG_RW_B;
						ELSIF(strcmp(ADR(straSplit[2]), ADR('R')) = 0)THEN
							pMapping.access:= DAV_CONFIG_RW_R;
						ELSE
							status:= 111;
						END_IF

						(* Area *)
						IF(strcmp(ADR(straSplit[3]), ADR('D')) = 0)THEN
							pMapping.var.area:= DAV_AREA_DB;
						ELSIF(strcmp(ADR(straSplit[3]), ADR('M')) = 0)THEN
							pMapping.var.area:= DAV_AREA_FLAG;
						ELSIF(strcmp(ADR(straSplit[3]), ADR('I')) = 0)THEN
							pMapping.var.area:= DAV_AREA_INPUT;
						ELSIF(strcmp(ADR(straSplit[3]), ADR('O')) = 0)THEN
							pMapping.var.area:= DAV_AREA_OUTPUT;
						ELSE
							status:= 112;
						END_IF

						(* DataBlock number *)
						IF(pMapping.var.area <> DAV_AREA_DB)THEN
							pMapping.var.db:= 0;
						ELSE
							IF(DAVisnumeric(ADR(straSplit[4])) = TRUE)THEN
								tmpVal:= atoi(ADR(straSplit[4]));

								IF((tmpVal >= 0) AND (tmpVal <= 65535))THEN
									pMapping.var.db:= DINT_TO_UINT(tmpVal);
								ELSE
									status:= 113;
								END_IF
							ELSE
								tmpAdr:= 0;
								curDataLength:= 0;
								status_i:= PV_xgetadr(ADR(straSplit[4]), ADR(tmpAdr), ADR(curDataLength));
								IF((status_i = 0) AND (tmpAdr <> 0) AND (curDataLength = 2))THEN
									pMapping.var.pdb:= tmpAdr;
								ELSE
									status:= 114;
								END_IF
							END_IF
						END_IF

						(* Start address (either value or variable) *)
						pMapping.var.pStartAdr:= 0;
						IF(DAVisnumeric(ADR(straSplit[5])) = TRUE)THEN
			 				pMapping.var.actAdr:= DINT_TO_UINT(atoi(ADR(straSplit[5])));
						ELSE
							(* User has included '+XX' *)
							posPlus:= INT_TO_UINT(FIND(straSplit[5], '+'));
							IF(posPlus > 0)THEN
								pMapping.var.actAdr:= DINT_TO_UINT(atoi(ADR(straSplit[5]) + posPlus));
								memset(ADR(straSplit[5]) + posPlus - 1, 0, SIZEOF(straSplit[0]) - posPlus + 1);
							ELSE
								pMapping.var.actAdr:= 0;
							END_IF
							tmpAdr:= 0;
							curDataLength:= 0;
							status_i:= PV_xgetadr(ADR(straSplit[5]), ADR(tmpAdr), ADR(curDataLength));
							IF((status_i = 0) AND (tmpAdr <> 0) AND (curDataLength = 2))THEN
								pMapping.var.pStartAdr:= tmpAdr;
								IF(posPlus > 0)THEN
									pMapping.var.pStartAdr:= pMapping.var.pStartAdr;
								END_IF
							ELSE
								status:= 115;
							END_IF
						END_IF

						(* Start address bit (either value or variable) *)
						pMapping.var.pStartAdrB:= 0;
						IF(DAVisnumeric(ADR(straSplit[6])) = TRUE)THEN
			 				tmpVal:= atoi(ADR(straSplit[6]));
							IF((tmpVal >= 0) AND (tmpVal <= 7))THEN
								pMapping.var.bitAdrB:= DINT_TO_USINT(tmpVal);
							ELSE
								status:= 116;
							END_IF
						ELSE
							tmpAdr:= 0;
							curDataLength:= 0;
							status_i:= PV_xgetadr(ADR(straSplit[6]), ADR(tmpAdr), ADR(curDataLength));
							IF((status_i = 0) AND (tmpAdr <> 0) AND (curDataLength = 1))THEN
								pMapping.var.pStartAdrB:= tmpAdr;
							ELSE
								status:= 117;
							END_IF
						END_IF

						(* Determine address in bits *)
						(* Note: if (pStartAdrXX > 0) then we need to keep recalculating this *)
						DAVcalcVARadr(ADR(pMapping.var));

						(* Length *)
						tmpVal:= atoi(ADR(straSplit[7]));
						IF((tmpVal = 1) OR (tmpVal = 2) OR (tmpVal = 4))THEN
			 				pMapping.var.length:= DINT_TO_USINT(tmpVal);
						ELSE
							status:= 118;
						END_IF

						(* B&R Variable *)
						tmpAdr:= 0;
						curDataLength:= 0;
						curDimensions:= 0;
						status_i:= PV_xgetadr(ADR(straSplit[8]), ADR(pMapping.brVarAdr), ADR(curDataLength));
						status_i:= status_i OR PV_ninfo(ADR(straSplit[8]), ADR(curVarType), ADR(curDataLength), ADR(curDimensions));
						IF((status_i = 0) AND ((curDataLength <= 4)) AND (pMapping.brVarAdr > 0))THEN
							pMapping.brVarType:= UDINT_TO_USINT(curVarType);						(* Store variable type *)
							pMapping.brVarLength:= UDINT_TO_USINT(curDataLength);				(* Store variable length *)
							memcpy(ADR(pMapping.brPrevValue), pMapping.brVarAdr, pMapping.brVarLength);		(* Store the previous value *)
						ELSE
							status:= 119;
						END_IF

						(* Variable type *)
						IF(pMapping.brVarType = 1)THEN
							pMapping.var.type:= DAV_VAR_BIT;
			 			ELSE
							pMapping.var.type:= DAV_VAR_BYTE;
						END_IF

						configIdx:= configIdx + 1;																	(* Use next configuration *)
						charIdx:= charIdx + posNextNull + 1;												(* Point to next line (nullIdx + 1) *)

						(* Reached number of configurations, or length of DataObject *)
						(* Note: Data Object aligns to 4 bytes *)
						IF((configIdx >= numItemsMapping) OR (charIdx >= DatObjInfo_Map.len - 4))THEN
							pDAV.maxLinesMapping:= configIdx;													(* Number of lines used *)
							state:= 40;
						END_IF
					ELSE
						status:= 120;
					END_IF

					(* Error occured *)
					IF(status <> 65535)THEN
						state:= 255;
					END_IF
				(************************************************************************************************************************)

				(************************************************************************************************************************)
				(* Free memory														                 																															*)
				(************************************************************************************************************************)
				40:
					IF pMemIdent = 0 THEN
						(* Free DRAM Memory *)
						status_i:= TMP_free(lengthToAllocate, pDOData);
					ELSE
						memFreeFB[1](enable:=1, ident:=pMemIdent, mem:=pDOData);
						status_i := memFreeFB[1].status;
						memHandle[1] := 0;
					END_IF

					(* Complete *)
					IF(status_i = 0)THEN
						state:= 50;

					(* Error *)
					ELSE
						status:= status_i;
						state:= 255;
					END_IF
				(************************************************************************************************************************)

				(************************************************************************************************************************)
				(* Allocate memory and assign offsets for Configuration Data																														*)
				(************************************************************************************************************************)
				50:
					(* Reset number of bytes to allocate *)
					lengthToAllocate:= 0;

					(* For all lines *)
					IF(pDAV.maxLinesConfig > 0)THEN
						FOR configIdx:=0 TO pDAV.maxLinesConfig-1 BY 1 DO
							pConfig ACCESS pDAV.pConfig + (configIdx * SIZEOF(pConfig));

							(* Increase memory size *)
							lengthToAllocate:= lengthToAllocate + pConfig.var.length;
						END_FOR
					END_IF

					IF pMemIdent = 0 THEN
						(* Create memory partition *)
						status_i:= TMP_alloc(lengthToAllocate, ADR(pDOData));
					ELSE
						memAllocFB[1](enable:=TRUE,	ident:=pMemIdent, len:=lengthToAllocate);
						status_i:=memAllocFB[1].status;
						IF status_i = 0 THEN
							memHandle[1] := memAllocFB[1].mem;
							pDOData := memAllocFB[1].mem;
						END_IF
					END_IF

					(* Complete *)
					IF(status_i = 0)THEN
						state:= 60;

						(* Clear memory *)
						memset(pDOData, 0, lengthToAllocate);

						(* For all lines *)
						IF(pDAV.maxLinesConfig > 0)THEN
							FOR configIdx:=0 TO pDAV.maxLinesConfig-1 BY 1 DO
								pConfig ACCESS pDAV.pConfig + (configIdx * SIZEOF(pConfig));

								(* Store memory address *)
								pConfig.brVarAdr:= pDOData;
								pDOData:= pDOData + pConfig.var.length;
							END_FOR
						END_IF

					(* Error *)
					ELSE
						status:= status_i;
						state:= 255;
					END_IF
				(************************************************************************************************************************)

				(************************************************************************************************************************)
				(* Organize structures		 								                 																															*)
				(************************************************************************************************************************)
				60:
					(* For all config lines *)
					IF(pDAV.maxLinesConfig > 1)THEN

						(* Organize via Priority *)
						FOR configIdx:=0 TO pDAV.maxLinesConfig-2 BY 1 DO
							pConfig ACCESS pDAV.pConfig + (configIdx * SIZEOF(pConfig));
							FOR orderIdx:=configIdx+1 TO pDAV.maxLinesConfig-1 BY 1 DO
								pConfigSwap ACCESS pDAV.pConfig + (orderIdx * SIZEOF(pConfig));

								(* Swap items *)
								IF(pConfig.priority > pConfigSwap.priority)THEN
				 					memcpy(ADR(configTemp), ADR(pConfig), SIZEOF(pConfig));
									memcpy(ADR(pConfig), ADR(pConfigSwap), SIZEOF(pConfig));
									memcpy(ADR(pConfigSwap), ADR(configTemp), SIZEOF(pConfig));
								END_IF
							END_FOR
						END_FOR

						(* Organize via Area *
						FOR configIdx:=0 TO pDAV.maxLinesConfig-2 BY 1 DO
							pConfig ACCESS pDAV.pConfig + (configIdx * SIZEOF(pConfig));
							FOR orderIdx:=configIdx+1 TO pDAV.maxLinesConfig-1 BY 1 DO
								pConfigSwap ACCESS pDAV.pConfig + (orderIdx * SIZEOF(pConfig));

								(* Swap items *
								IF((pConfig.priority = pConfigSwap.priority) AND
									(pConfig.var.area = DAV_AREA_DB) AND (pConfigSwap.var.area <> DAV_AREA_DB))THEN
					 					memcpy(ADR(configTemp), ADR(pConfig), SIZEOF(pConfig));
										memcpy(ADR(pConfig), ADR(pConfigSwap), SIZEOF(pConfig));
										memcpy(ADR(pConfigSwap), ADR(configTemp), SIZEOF(pConfig));
								END_IF
							END_FOR
						END_FOR

						(* Organize via DataBlock *
						FOR configIdx:=0 TO pDAV.maxLinesConfig-2 BY 1 DO
							pConfig ACCESS pDAV.pConfig + (configIdx * SIZEOF(pConfig));
							FOR orderIdx:=configIdx+1 TO pDAV.maxLinesConfig-1 BY 1 DO
								pConfigSwap ACCESS pDAV.pConfig + (orderIdx * SIZEOF(pConfig));

								(* Swap items *
								IF((pConfig.priority = pConfigSwap.priority) AND
									(pConfig.var.area = DAV_AREA_DB) AND (pConfigSwap.var.area = DAV_AREA_DB) AND
									(pConfig.var.db > pConfigSwap.var.db))THEN
					 					memcpy(ADR(configTemp), ADR(pConfig), SIZEOF(pConfig));
										memcpy(ADR(pConfig), ADR(pConfigSwap), SIZEOF(pConfig));
										memcpy(ADR(pConfigSwap), ADR(configTemp), SIZEOF(pConfig));
								END_IF
							END_FOR
						END_FOR

						(* Organize via Start Address *
						FOR configIdx:=0 TO pDAV.maxLinesConfig-2 BY 1 DO
							pConfig ACCESS pDAV.pConfig + (configIdx * SIZEOF(pConfig));
							FOR orderIdx:=configIdx+1 TO pDAV.maxLinesConfig-1 BY 1 DO
								pConfigSwap ACCESS pDAV.pConfig + (orderIdx * SIZEOF(pConfig));

								(* Swap items *
								IF((pConfig.priority = pConfigSwap.priority) AND
									(pConfig.var.area = pConfigSwap.var.area) AND
									(pConfig.var.db = pConfigSwap.var.db) AND
									(pConfig.var.bitAdr > pConfigSwap.var.bitAdr))THEN
					 					memcpy(ADR(configTemp), ADR(pConfig), SIZEOF(pConfig));
										memcpy(ADR(pConfig), ADR(pConfigSwap), SIZEOF(pConfig));
										memcpy(ADR(pConfigSwap), ADR(configTemp), SIZEOF(pConfig));
								END_IF
							END_FOR
						END_FOR
						*)
					END_IF

					(* For all mapping lines *)
					IF(pDAV.maxLinesMapping > 1)THEN

						(* Organize via Priority *)
						FOR configIdx:=0 TO pDAV.maxLinesMapping-2 BY 1 DO
							pMapping ACCESS pDAV.pMapping + (configIdx * SIZEOF(pMapping));
							FOR orderIdx:=configIdx+1 TO pDAV.maxLinesMapping-1 BY 1 DO
								pMappingSwap ACCESS pDAV.pMapping + (orderIdx * SIZEOF(pMapping));

								(* Swap items *)
								IF(pMapping.priority > pMappingSwap.priority)THEN
				 					memcpy(ADR(mappingTemp), ADR(pMapping), SIZEOF(pMapping));
									memcpy(ADR(pMapping), ADR(pMappingSwap), SIZEOF(pMapping));
									memcpy(ADR(pMappingSwap), ADR(mappingTemp), SIZEOF(pMapping));
								END_IF
							END_FOR
						END_FOR

						(* Organize via Access *)
						FOR configIdx:=0 TO pDAV.maxLinesMapping-2 BY 1 DO
							pMapping ACCESS pDAV.pMapping + (configIdx * SIZEOF(pMapping));
							FOR orderIdx:=configIdx+1 TO pDAV.maxLinesMapping-1 BY 1 DO
								pMappingSwap ACCESS pDAV.pMapping + (orderIdx * SIZEOF(pMapping));

								(* Swap items *)
								IF((pMapping.priority = pMappingSwap.priority) AND
									(pMapping.access < pMappingSwap.access))THEN
				 					memcpy(ADR(mappingTemp), ADR(pMapping), SIZEOF(pMapping));
									memcpy(ADR(pMapping), ADR(pMappingSwap), SIZEOF(pMapping));
									memcpy(ADR(pMappingSwap), ADR(mappingTemp), SIZEOF(pMapping));
								END_IF
							END_FOR
						END_FOR
					END_IF

					(* Complete *)
					state:= 61;
				(************************************************************************************************************************)

				(************************************************************************************************************************)
				(* Store Configuration Index							                 																															*)
				(* Used so we don't replicate the same READ data when sending packets																										*)
				(************************************************************************************************************************)
				61:
					(* For all mapping lines *)
					IF((pDAV.maxLinesMapping > 0) AND (pDAV.maxLinesConfig > 0))THEN
						FOR mappingIdx:=0 TO pDAV.maxLinesMapping-1 BY 1 DO
							pMapping ACCESS pDAV.pMapping + (mappingIdx * SIZEOF(pMapping));
							FOR configIdx:=0 TO pDAV.maxLinesConfig-1 BY 1 DO
								pConfig ACCESS pDAV.pConfig + (configIdx * SIZEOF(pConfig));

								(* Store configuration index if mapping variable fits *)
									IF((pMapping.var.area = pConfig.var.area) AND
										(pMapping.var.db = pConfig.var.db) AND
										(pMapping.var.pdb = pConfig.var.pdb) AND
										(pMapping.var.pStartAdr = pConfig.var.pStartAdr) AND
										(pMapping.var.bitAdr >= pConfig.var.bitAdr) AND
										(pMapping.var.bitAdr + SEL((pMapping.var.type = DAV_VAR_BIT), (pMapping.var.length * 8), 1) <=
											pConfig.var.bitAdr + SEL((pConfig.var.type = DAV_VAR_BIT), (pConfig.var.length * 8), 1)))THEN
									pMapping.cfgIndex:= configIdx;
								END_IF
							END_FOR
						END_FOR
					END_IF

					(* Complete *)
					state:= 200;
					status:= 0;
					pDAV.internal:= 1;
				(************************************************************************************************************************)

				(************************************************************************************************************************)
				(* Complete										  					                 																															*)
				(************************************************************************************************************************)
				200:
					IF reset THEN
						status := 65535;
						state := 0;
					END_IF

				(************************************************************************************************************************)

				(************************************************************************************************************************)
				(* Error										  					                 																																*)
				(************************************************************************************************************************)
				255:
					IF reset THEN
						status := 65535;
						state := 0;
					END_IF
				(************************************************************************************************************************)

			END_CASE
			(**************************************************************************************************************************)
			(* End of Function Operation                                                            																	*)
			(**************************************************************************************************************************)

			(**************************************************************************************************************************)
			(* Check scan count 																																																			*)
			(**************************************************************************************************************************)
			scanCount:= scanCount + 1;																				(* Increase scan count *)
			IF((status = 65535) AND (scanCount > 100000))THEN
	 			status:= DAV_ERR_CFG_TIMEOUT;																		(* Exit while if the scanCount is too large *)
	 		END_IF
			(**************************************************************************************************************************)

	END_IF

END_FUNCTION_BLOCK
(********************************************************************************************************************************)
(* End of DAVinitialize																																																					*)
(********************************************************************************************************************************)
```

#### DAVconnection.st - Connects / Disconnects to a PLC
```iecst
(********************************************************************************************************************************)
(* COPYRIGHT -- B&R Industrial Automation																																												*)
(********************************************************************************************************************************)
(* Library:				DAVNoDave																																																			*)
(* File: 					DAVconnection.st																																															*)
(* Author: 				morrisd																																																				*)
(* Created: 			May 26, 2009																																																	*)
(********************************************************************************************************************************)

(********************************************************************************************************************************)
(* DAVconnect																																																										*)
(*==============================================================================================================================*)
(* Creates a connection to the Siemen's PLC		 																																									*)
(* Returns the status and a handle used for the other DAVxx functions																														*)
(********************************************************************************************************************************)
FUNCTION_BLOCK DAVconnect

	(* Function not enabled *)
	IF(enable = FALSE)THEN
		status:= 65534;

	(* Invalid handle *)
	ELSIF(pHandle = 0)THEN
 		status:= DAV_ERR_HANDLE;

	(* Invalid connection *)
	ELSIF((protocol <> DAV_PROTOCOL_TCP) AND (protocol <> DAV_PROTOCOL_MPI))THEN
		status:= DAV_ERR_CONNECT_PROTOCOL;

	(* Invalid interface *)
	ELSIF((protocol = DAV_PROTOCOL_MPI) AND (pMPIinterface = 0))THEN
 		status:= DAV_ERR_CONNECT_INTERFACE;

	(* Invalid IP address *)
	ELSIF((protocol = DAV_PROTOCOL_TCP) AND (pTCPtargetIP = 0))THEN
 		status:= DAV_ERR_CONNECT_TARGETIP;

	(* Run the function *)
	ELSE

		(* Make status busy *)
		status:= 65535;

		(****************************************************************************************************************************)
		(* Map data (to avoid errors if the user changes them during operation                  																		*)
		(****************************************************************************************************************************)
		IF(state = 0)THEN

			(* Reset PDU Length *)
			pduLength:= 0;
			portOpened:= 0;

			(* Access handle *)
			pDAV ACCESS pHandle;

			(* Access buffer *)
			pBufferR ACCESS pDAV.pBufferR;
			memset(pDAV.pBufferR, 0, DAV_DEFAULT_BUFFER_R);

			(* Valid configuration *)
			IF((pDAV.ident = 0) AND (pDAV.connection.protocol = 0) AND
			(pDAV.pBufferR <> 0) AND (pDAV.pBufferW <> 0))THEN

				(* Internal *)
				memset(ADR(pDAV.connection), 0, SIZEOF(pDAV.connection));
				pDAV.connection.protocol:=		protocol;									(* Store protocol *)
				pDAV.connection.mpiSpeed:=		MPIspeed;									(* Store MPI speed *)
				pDAV.connection.mpiLocalAdr:=	MPIlocalAdr;							(* Store MPI local address *)
				pDAV.connection.mpiPLCAdr:=		MPIplcAdr;								(* Store MPI PLC address *)
				pDAV.connection.tcpRack:=			TCPrack;									(* Store TCP rack *)
				pDAV.connection.tcpSlot:=			TCPslot;									(* Store TCP slot *)
				pDAV.connection.connectNum:=	16#14;										(* Connection number *)
				pDAV.connection.connectNum2:=	16#03;										(* Connection number 2 (what it should be) *)
				pDAV.connection.pduNum:=			16#FFFE;									(* PDU number *)
				pDAV.connection.msgNum:=			16#00;										(* Message number *)

				(* Initialize DAVsend *)
				DAVexchange_0.enable:=				TRUE;											(* Enable function block *)
				DAVexchange_0.pHandle:=				pHandle;									(* Handle from DAVinitialize *)
				DAVexchange_0.sendLength:=		0;												(* Size of sending data - calculated later *)
				DAVexchange_0.mpiFullExchange:=		FALSE;								(* Disable full packet exchange *)

				(* Determine timeout *)
				IF(timeout = DAV_DEFAULT_TIMEOUT)THEN
					IF(pDAV.connection.protocol = DAV_PROTOCOL_TCP)THEN
						DAVexchange_0.timeout:=		150;											(* 1500ms *)
					ELSE
						DAVexchange_0.timeout:=		500;											(* 5000ms *)
					END_IF
				ELSE
					DAVexchange_0.timeout:=			timeout;									(* User's timeout *)
				END_IF

				(* Initialize TCP comms *)
				IF(pDAV.connection.protocol = DAV_PROTOCOL_TCP)THEN

					(* Initialize TcpOpen function block *)
	 				TcpOpen_0.enable:=					TRUE;									(* Enable function block *)
					TcpOpen_0.pIfAddr:= 				pTCPsourceIP;							(* IP Address of port to use *)
					TcpOpen_0.options:= 				0;										(* Default options *)

					IF(TcpOpen_0.port = 0)THEN
						TcpOpen_0.port:=					DAV_DEFAULT_SOURCE_PORT;	(* Use an dynamic port (49152 < port < 65535) *)
					ELSE
						TcpOpen_0.port:=					TcpOpen_0.port + 1;				(* Use next port *)
					END_IF

					(* Initialize TcpClient function block *)
	 				TcpClient_0.enable:= 				TRUE;											(* Enable function block *)
					TcpClient_0.pServer:= 			pTCPtargetIP;							(* Siemens IP Address *)
					IF(TCPport = 0)THEN
						TcpClient_0.portserv:=		DAV_DEFAULT_PORT;					(* Use default port *)
					ELSE
						TcpClient_0.portserv:=		TCPport;									(* Use users port *)
					END_IF

					(* Initialize TON_10ms function block *)
					TON_10ms_ClientTimeout.IN:=	FALSE;										(* Turn timer off *)
					TON_10ms_ClientTimeout.PT:= 500;											(* 5 seconds timeout *)
					TON_10ms_ClientTimeout();															(* Call function to reset timer *)
					TON_10ms_ClientTimeout.IN:= TRUE;											(* Enable timer *)

					(* TCP initialize state *)
					state:= 100;

				(* Initialize MPI comms *)
				ELSIF(pDAV.connection.protocol = DAV_PROTOCOL_MPI)THEN

					(* Initialize XOPENCONFIG structure *)
					frmConfig.idle:=						4;												(* Idle time between characters: 50ms/38700 = 150 *)
					frmConfig.delimc:=					0;												(* Number of delimiter characters *)
					frmConfig.delim[0]:=				0;												(* Delimiter character *)
					frmConfig.delim[1]:=				0;												(* Delimiter character *)
					frmConfig.tx_cnt:=					2;												(* Number of transmit buffers *)
					frmConfig.rx_cnt:=					2;												(* Number of receive buffers *)
					frmConfig.tx_len:=					DAV_PDU_SIZE + 20;				(* Transmit buffer length *)
					frmConfig.rx_len:=					DAV_PDU_SIZE + 20;				(* Receive buffer length *)
					frmConfig.argc:=						0;												(* Number of additional arguments *)
					frmConfig.argv:=						0;												(* Address of additional arguments *)

					(* Initialize FRM_XOpen function block *)
					FRM_xopen_0.enable:=				TRUE;											(* Enable function block *)
					FRM_xopen_0.device:=				pMPIinterface;						(* Interface to use *)
					IF(pMPIconnection <> 0)THEN
						FRM_xopen_0.mode:= 				pMPIconnection;						(* Users connection parameter *)
					ELSE
						FRM_xopen_0.mode:= 				ADR(DAV_DEFAULT_MPI);			(* Use default connection *)
					END_IF
					FRM_xopen_0.config:= 				ADR(frmConfig);						(* Pointer to configuration *)

					(* MPI initialize state *)
					state:= 200;
				END_IF

			(* Connection already open *)
			ELSIF((pDAV.ident <> 0) OR (pDAV.connection.protocol <> 0))THEN
				status:= DAV_ERR_CONNECT_OPEN;

			(* Invalid configuration *)
			ELSE
				status:= DAV_ERR_INITIALIZATION;
			END_IF
		END_IF
		(****************************************************************************************************************************)

		(****************************************************************************************************************************)
		(* Function Operation                                                                     																	*)
		(****************************************************************************************************************************)
		CASE state OF

			(**************************************************************************************************************************)
			(* Open Port                                                                            																	*)
			(**************************************************************************************************************************)
			100:
				(* Service function *)
				TcpOpen_0();

				(* Port opened *)
				IF(TcpOpen_0.status = 0)THEN
					pDAV.ident:=							TcpOpen_0.ident;
					TcpClient_0.ident:= 					TcpOpen_0.ident;
					TCPident := 							TcpOpen_0.ident;
					portOpened:=							TcpOpen_0.port;
					state:= 101;

				(* Port already open, use next port number *)
				ELSIF(TcpOpen_0.status = tcpERR_ALREADY_EXIST)THEN
					TcpOpen_0.port:= 					TcpOpen_0.port + 1;

				(* Error *)
				ELSIF(TcpOpen_0.status <> 65535)THEN
					status:= TcpOpen_0.status;
				END_IF
			(**************************************************************************************************************************)

			(**************************************************************************************************************************)
			(* Connect to Siemens PLC                                                               																	*)
			(**************************************************************************************************************************)
			101:
				(* Service function *)
				TcpClient_0();

				(* Service timeout *)
				TON_10ms_ClientTimeout();

				(* Client connected *)
				IF(TcpClient_0.status = 0)THEN

					(* Build up packet - connect to PLC *)
					memset(pDAV.pBufferW, 0, DAV_DEFAULT_BUFFER_W);
					DAVexchange_0.sendLength:= DAVpacketTCPconnect(pHandle, pDAV.pBufferW, 0);
					state:= 102;

				(* Timeout *)
				ELSIF(TON_10ms_ClientTimeout.Q)THEN
					status:= DAV_ERR_CONNECT_TCP;

				(* Error *)
				ELSIF(TcpClient_0.status <> 65535)THEN
					status:= TcpClient_0.status;
				END_IF
			(**************************************************************************************************************************)

			(**************************************************************************************************************************)
			(* Send connection block and get it's response                                          																	*)
			(**************************************************************************************************************************)
			102:
				(* Service function *)
				DAVexchange_0();

				(* Data sent and received *)
				IF(DAVexchange_0.status = 0)THEN

					(* Build up packet - get PDU size *)
					memset(pDAV.pBufferW, 0, DAV_DEFAULT_BUFFER_W);
					DAVexchange_0.sendLength:= DAVpacketTCPconnect(pHandle, pDAV.pBufferW, 1);
					state:= 103;

				(* Error *)
				ELSIF(DAVexchange_0.status <> 65535)THEN
					status:= DAVexchange_0.status;
				END_IF
			(**************************************************************************************************************************)

			(**************************************************************************************************************************)
			(* Send PDU block and get it's response                                                 																	*)
			(**************************************************************************************************************************)
			103:
				(* Service function *)
				DAVexchange_0();

				(* Data sent and received *)
				IF(DAVexchange_0.status = 0)THEN

					(* Get PDU Length *)
					memcpy(ADR(pduLength), pDAV.pBufferR + DAVexchange_0.recvStartOfDataIdx, 1);

					(* Initialize Client *)
					status:= 0;

				(* Error *)
				ELSIF(DAVexchange_0.status <> 65535)THEN
					status:= DAVexchange_0.status;
				END_IF
			(**************************************************************************************************************************)

			(**************************************************************************************************************************)
			(* Open interface												                                                																	*)
			(**************************************************************************************************************************)
			200:
				(* Service function *)
				FRM_xopen_0();

				(* Data sent and received *)
				IF(FRM_xopen_0.status = 0)THEN
					pDAV.ident:= FRM_xopen_0.ident;

					(* Build up packet - get MPI adapter version (1) *)
					memset(pDAV.pBufferW, 0, DAV_DEFAULT_BUFFER_W);
					DAVexchange_0.sendLength:= DAVpacketMPIconnect(pHandle, pDAV.pBufferW, 0);
					state:= 201;

				(* Error *)
				ELSIF(FRM_xopen_0.status <> 65535)THEN
					status:= FRM_xopen_0.status;
				END_IF
			(**************************************************************************************************************************)

			(**************************************************************************************************************************)
			(* Send packet to get the MPI adapter version and get it's response (1)                  																	*)
			(**************************************************************************************************************************)
			201:
				(* Service function *)
				DAVexchange_0();

				(* Data sent and received *)
				IF(DAVexchange_0.status = 0)THEN

					(* Check response *)
					IF((DAVexchange_0.recvLength = 12) AND
						(DAVmpiCalcCS(pDAV.pBufferR, DAVexchange_0.recvLength) = TRUE) AND
						(DAVresponseMPIconnect(ADR(pDAV), pDAV.pBufferR, 0) = TRUE))THEN

						(* Build up packet - get MPI adapter version (2) *)
						memset(pDAV.pBufferW, 0, DAV_DEFAULT_BUFFER_W);
						DAVexchange_0.sendLength:= DAVpacketMPIconnect(pHandle, pDAV.pBufferW, 1);
						state:= 202;

		 			(* Invalid response *)
		 			ELSE
						status:= DAV_ERR_RECV_RESPONSE;
					END_IF

				(* Error *)
				ELSIF(DAVexchange_0.status <> 65535)THEN
					status:= DAVexchange_0.status;
				END_IF
			(**************************************************************************************************************************)

			(**************************************************************************************************************************)
			(* Send packet to get the MPI adapter version and get it's response (2)                  																	*)
			(**************************************************************************************************************************)
			202:
				(* Service function *)
				DAVexchange_0();

				(* Data sent and received *)
				IF(DAVexchange_0.status = 0)THEN

					(* Check response *)
					IF((DAVexchange_0.recvLength = 12) AND
						(DAVmpiCalcCS(pDAV.pBufferR, DAVexchange_0.recvLength) = TRUE) AND
						(DAVresponseMPIconnect(ADR(pDAV), pDAV.pBufferR, 1) = TRUE))THEN

						(* Build up packet - connect to PLC (1) *)
						memset(pDAV.pBufferW, 0, DAV_DEFAULT_BUFFER_W);
						DAVexchange_0.sendLength:= DAVpacketMPIconnect(pHandle, pDAV.pBufferW, 2);
						state:= 203;

		 			(* Invalid MPI adapter - perhaps adapter0330 *)
					ELSE
						status:= DAV_ERR_MPI_ADAPTER;
					END_IF

				(* Error *)
				ELSIF(DAVexchange_0.status <> 65535)THEN
					status:= DAVexchange_0.status;
				END_IF
			(**************************************************************************************************************************)

			(**************************************************************************************************************************)
			(* Send packet to connect to the PLC and get it's response (1)                          																	*)
			(**************************************************************************************************************************)
			203:
				(* Service function *)
				DAVexchange_0();

				(* Data sent and received *)
				IF(DAVexchange_0.status = 0)THEN

					(* Check response *)
					IF((DAVexchange_0.recvLength = 21) AND
						(DAVmpiCalcCS(pDAV.pBufferR, DAVexchange_0.recvLength) = TRUE) AND
						(DAVresponseMPIconnect(ADR(pDAV), pDAV.pBufferR, 2) = TRUE))THEN

						(* Update connection packet *)
						pDAV.connection.connectNum2:= pBufferR[5];

						(* Build up packet - connect to PLC (2) *)
						memset(pDAV.pBufferW, 0, DAV_DEFAULT_BUFFER_W);
						DAVexchange_0.sendLength:= DAVpacketMPIconnect(pHandle, pDAV.pBufferW, 3);
						state:= 204;

		 			(* Invalid response *)
		 			ELSE
						status:= DAV_ERR_RECV_RESPONSE;
					END_IF

				(* Error *)
				ELSIF(DAVexchange_0.status <> 65535)THEN
					status:= DAVexchange_0.status;
				END_IF
			(**************************************************************************************************************************)

			(**************************************************************************************************************************)
			(* Send packet to connect to the PLC and get it's response (2)                          																	*)
			(**************************************************************************************************************************)
			204:
				(* Service function *)
				DAVexchange_0();

				(* Data sent and received *)
				IF(DAVexchange_0.status = 0)THEN

						(* Check response *)
					IF((DAVexchange_0.recvLength = 11) AND
						(DAVmpiCalcCS(pDAV.pBufferR, DAVexchange_0.recvLength) = TRUE) AND
						(DAVresponseMPIconnect(ADR(pDAV), pDAV.pBufferR, 3) = TRUE))THEN

						(* Build up packet - get PDU length *)
						memset(pDAV.pBufferW, 0, DAV_DEFAULT_BUFFER_W);
						DAVexchange_0.sendLength:= DAVpacketMPIconnect(pHandle, pDAV.pBufferW, 4);
						state:= 205;

					(* Invalid MPI adapter - perhaps adapter0330 *)
					ELSE
						status:= DAV_ERR_RECV_PROTOCOL;
					END_IF
				(* Error *)
				ELSIF(DAVexchange_0.status <> 65535)THEN
					status:= DAVexchange_0.status;
				END_IF
			(**************************************************************************************************************************)

			(**************************************************************************************************************************)
			(* Send connection block and get it's response PDU                                         																*)
			(**************************************************************************************************************************)
			205:
				(* Service function *)
				DAVexchange_0.mpiFullExchange:=	TRUE;
				DAVexchange_0();

				(* Data sent and received *)
				IF(DAVexchange_0.status = 0)THEN

					(* Get PDU Length *)
					pduLength:= DAVswapWORD(pDAV.pBufferR + DAVexchange_0.recvStartOfDataIdx + 6);

					(* Initialize Client *)
					status:= 0;

				(* Error *)
				ELSIF(DAVexchange_0.status <> 65535)THEN
					status:= DAVexchange_0.status;
				END_IF
			(**************************************************************************************************************************)
		END_CASE

		(* Return to Initialization state *)
		IF(status <> 65535)THEN
			IF(status = 0)THEN
	 			pDAV.internal:= 2;
			END_IF
			state:= 0;
		END_IF
		(****************************************************************************************************************************)
		(* End of Function Operation                                                              																	*)
		(****************************************************************************************************************************)

	END_IF
END_FUNCTION_BLOCK
(********************************************************************************************************************************)
(* End of DAVconnect																																																						*)
(********************************************************************************************************************************)

(********************************************************************************************************************************)
(* DAVdisconnect																																																								*)
(*==============================================================================================================================*)
(* Disconnects the current connection to the Siemen's PLC		 																																		*)
(* Returns the status 																																																					*)
(********************************************************************************************************************************)
FUNCTION_BLOCK DAVdisconnect

	(* Function not enabled *)
	IF(enable = FALSE)THEN
		status:= 65534;

	(* Invalid handle *)
	ELSIF(pHandle = 0)THEN
 		status:= DAV_ERR_HANDLE;

	(* Run the function *)
	ELSE

		(* Make status busy *)
		status:= 65535;

		(****************************************************************************************************************************)
		(* Map data (to avoid errors if the user changes them during operation                 																			*)
		(****************************************************************************************************************************)
		IF(state = 0)THEN

			(* Access handle *)
			pDAV ACCESS pHandle;

			(* Initialize DAVsend function block *)
			DAVexchange_0.enable:=							TRUE;											(* Enable function block *)
			DAVexchange_0.pHandle:=							pHandle;									(* Handle from DAVinitialize *)
			DAVexchange_0.sendLength:=					0;												(* Size of sending data - calculated later *)
			DAVexchange_0.mpiFullExchange:=			FALSE;										(* Disable full packet exchange *)

			(* Determine timeout *)
			IF(timeout = DAV_DEFAULT_TIMEOUT)THEN
				IF(pDAV.connection.protocol = DAV_PROTOCOL_TCP)THEN
					DAVexchange_0.timeout:=					150;											(* 1500ms *)
				ELSE
					DAVexchange_0.timeout:=					500;											(* 5000ms *)
				END_IF
			ELSE
				DAVexchange_0.timeout:=						timeout;									(* User's timeout *)
			END_IF

			(* Create Disconnect packet (0) *)
			memset(pDAV.pBufferW, 0, DAV_DEFAULT_BUFFER_W);
			DAVexchange_0.sendLength:= DAVpacketMPIdisconnect(pHandle, pDAV.pBufferW, 0);

			(* Initialize TcpClose function block *)
			TcpClose_0.enable:=							TRUE;											(* Enable function block *)
			TcpClose_0.ident:=							pDAV.ident;										(* TcpOpen ident *)
			TcpClose_0.how:=							0;												(* Close all communcations *)

			(* Initialize FRM_close function block *)
			FRM_close_0.enable:=						TRUE;											(* Enable function block *)
			FRM_close_0.ident:=							pDAV.ident;								(* FRM_Xopen ident *)

			(* Close TCP comms *)
			IF(pDAV.connection.protocol = DAV_PROTOCOL_TCP)THEN
				state:= 100;

			(* Close MPI comms *)
			ELSIF(pDAV.connection.protocol = DAV_PROTOCOL_MPI)THEN
				state:= 200;

			(* Invalid mode *)
			ELSE
				status:= DAV_ERR_CONNECT_CLOSED;
			END_IF
		END_IF
		(****************************************************************************************************************************)

		(****************************************************************************************************************************)
		(* Function Operation                                                                     																	*)
		(****************************************************************************************************************************)
		CASE state OF

			(**************************************************************************************************************************)
			(* Close Port                                                                            																	*)
			(**************************************************************************************************************************)
			100:
				(* Service function *)
				TcpClose_0();

				(* Port opened *)
				IF(TcpClose_0.status = 0)THEN
					status:= 0;

				(* Error *)
				ELSIF(TcpClose_0.status <> 65535)THEN
					status:= TcpClose_0.status;
				END_IF
			(**************************************************************************************************************************)

			(**************************************************************************************************************************)
			(* Disconnect from the PLC                                                              																	*)
			(**************************************************************************************************************************)
			200:
				(* Service function *)
				DAVexchange_0();

				(* Data sent and received *)
				IF(DAVexchange_0.status = 0)THEN

					(* Create Disconnect packet (0) *)
					memset(pDAV.pBufferW, 0, DAV_DEFAULT_BUFFER_W);
					DAVexchange_0.sendLength:= DAVpacketMPIdisconnect(pHandle, pDAV.pBufferW, 1);
					state:= 201;

				(* Error *)
				ELSIF(DAVexchange_0.status <> 65535)THEN
					status:= DAVexchange_0.status;
				END_IF

			(**************************************************************************************************************************)

			(**************************************************************************************************************************)
			(* Disconnect from the MPI Adapter                                                       																	*)
			(**************************************************************************************************************************)
			201:
				(* Service function *)
				DAVexchange_0();

				(* Data sent and received *)
				IF(DAVexchange_0.status = 0)THEN
					state:= 202;

				(* Error *)
				ELSIF(DAVexchange_0.status <> 65535)THEN
					status:= DAVexchange_0.status;
				END_IF

			(**************************************************************************************************************************)

			(**************************************************************************************************************************)
			(* Close Port                                                                            																	*)
			(**************************************************************************************************************************)
			202:
				(* Service function *)
				FRM_close_0();

				(* Port opened *)
				IF(FRM_close_0.status = 0)THEN
					status:= 0;

				(* Error *)
				ELSIF(FRM_close_0.status <> 65535)THEN
					status:= FRM_close_0.status;
				END_IF
			(**************************************************************************************************************************)
		END_CASE

		(* Return to Initialization state *)
		IF(status <> 65535)THEN

			(* Reconnection required *)
			IF(status = 0)THEN
				IF(pDAV.internal > 1)THEN
	 				pDAV.internal:= 1;
				END_IF
				pDAV.ident:= 0;
				memset(ADR(pDAV.connection), 0, SIZEOF(pDAV.connection));
			END_IF
			state:= 0;
		END_IF
		(****************************************************************************************************************************)
		(* End of Function Operation                                                               																	*)
		(****************************************************************************************************************************)
	END_IF
END_FUNCTION_BLOCK
(********************************************************************************************************************************)
(* End of DAVdisconnect																																																					*)
(********************************************************************************************************************************)
```
